(* IEC 61131-3 sources: CodesysTest/alpha/export/Device.dev/Plc Logic/Application/FBs/Components/FunnelFB.pou/DelaySetting.prop, 1 file *)

(* ---- Get.pm.st ---- *)
(*#-#-#-#-#-#-#-#-#-#---Declaration---#-#-#-#-#-#-#-#-#-#-#-#-#*)

VAR
END_VAR
(*#-#-#-#-#-#-#-#-#-#---Implementation---#-#-#-#-#-#-#-#-#-#-#-#-#*)

DelaySetting := TO_REAL(openDelayTimer.PT ) / 1000;
